// TIA Portal project "PLC and HMI project in TIA Portal.- simple" (V20)

(* hardware
DEVICE "S7-1200 station_1"  S7-1200 Station
   slot 0: "Rack_0"  S7-1200 Rack  Rack  V1.0
   slot 1: "PLC_1"  CPU 1212FC DC/DC/DC  6ES7 212-1AF40-0XB0  V4.7
DEVICE "HMI_1"  KTP700 Basic PN
   slot 0: "HMI_1"  KTP700 Basic PN  6AV2 123-2GB03-0AX0  17.0.0.0
   slot 1: "HMI_RT_1"  KTP700 Basic PN  6AV2 123-2GB03-0AX0  17.0.0.0
   slot 5: "HMI_1.IE_CP_1"  PROFINET Interface  17.0.0.0
      slot 1: "PROFINET Interface_1"  PROFINET Interface
         slot 1: "Port_1"  Port
*)

// ===== PLC "PLC_1"  CPU 1212FC DC/DC/DC =====

VAR_GLOBAL   // PLC tag table "Tag table_1"
   "Start_PB" AT %I0.0 : Bool;
   "Stop_PB" AT %M0.1 : Bool;
   "E_Stop" AT %M0.2 : Bool;
   "Conveyor_Motor" AT %Q0.0 : Bool;
END_VAR

DATA_BLOCK "Main_Safety_RTG1_DB"   // DB1, F_DB
{ S7_Optimized_Access := 'TRUE' }
NAME : FUSI
VERSION : 0.1
// stored: InstanceOfName Main_Safety_RTG1
"Main_Safety_RTG1"
BEGIN
END_DATA_BLOCK

FUNCTION_BLOCK "Main_Safety_RTG1"   // FB1, F_FBD
{ S7_Optimized_Access := 'TRUE' }
BEGIN
END_FUNCTION_BLOCK

ORGANIZATION_BLOCK "Main"   // OB1, LAD, ProgramCycle
TITLE = "Main Program Sweep (Cycle)"
{ S7_Optimized_Access := 'TRUE' }
VERSION : 0.1
   VAR_INPUT
      Initial_Call : Bool;   // Initial call of this OB
      Remanence : Bool;   // =True, if remanent data are available
   END_VAR
   VAR_TEMP   // added for the SCL form of the ladder/FBD networks
      _w1 : Bool;
   END_VAR
BEGIN

REGION Network 1
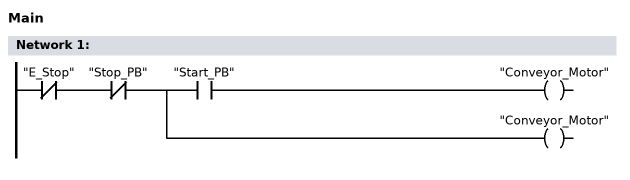
   RUNG wire#powerrail
      I_Contact( "E_Stop" )
      I_Contact( "Stop_PB" )
      wire#w1
      Contact( "Start_PB" )
      Coil( "Conveyor_Motor" )
   END_RUNG
   RUNG wire#w1
      Coil( "Conveyor_Motor" )
   END_RUNG
   // the same network as SCL:
   #_w1 := NOT "E_Stop" AND NOT "Stop_PB";
   "Conveyor_Motor" := #_w1 AND "Start_PB";
   "Conveyor_Motor" := #_w1;
END_REGION
END_ORGANIZATION_BLOCK

(* ===== HMI "HMI_RT_1" =====
system functions are stored by id; their names below are inferred from use
connection "HMI_Connection_1": ETHERNET, SMART_S7_1200_OMS

HMI tags "Default tag table"
   "Tag_ScreenNumber" : UInt, internal
   "Start_PB" : Bool = PLC Start_PB AT %I0.0, 1 s
   "Stop_PB" : Bool = PLC Stop_PB AT %M0.1, 1 s
   "E_Stop" : Bool = PLC E_Stop AT %M0.2, 1 s
   "Conveyor_Motor" : Bool = PLC Conveyor_Motor AT %Q0.0, 1 s

Template "Template_1" 800x480
   Button "Exit" at 714,429 size 71x50; TextOff 'Exit'; PictureOff "ExitRuntime_KTP700_Basic_PN_TR"; PictureOn "ExitRuntime_KTP700_Basic_PN_TR"
      on Release: StopRuntime(0)
   Button "Template_Button" at 614,429 size 71x50; TextOff 'Text'
   Button "Template_Button_1" at 514,429 size 71x50; TextOff 'Text'
   Button "Template_Button_2" at 414,429 size 71x50; TextOff 'Text'
   Button "Template_Button_3" at 314,429 size 71x50; TextOff 'Text'
   Button "Template_Button_4" at 214,429 size 71x50; TextOff 'Text'
   Button "Template_Button_5" at 114,429 size 71x50; TextOff 'Text'
   Button "Start screen" at 14,429 size 71x50; TextOff 'Start screen'; PictureOff "NavigateHome_KTP700_Basic_PN_TR"; PictureOn "NavigateHome_KTP700_Basic_PN_TR"
      on Release: ActivateScreen("Root screen", 0)
   SymbolicIOField "Symbolic_IO_Field_Screen" at 93,9 size 600x33; TextOff '0'; TextOn '1'; TextList "TextList_ScreenNames"
      ProcessValue <- "Tag_ScreenNumber"
      on Change: ActivateScreenByNumber("Tag_ScreenNumber", 0)
   DateTimeField "HmiScreenItemData" at 695,25 size 105x25
   DateTimeField "HmiScreenItemData_1" at 695,0 size 105x25
   GraphicView "Logo" at 0,0 size 91x51; Picture "Logo of HMI_1"

screen "Root screen" 800x480, template "Template_1"
   on GenerateScreen: SetTag("Stop_PB", 1)
   Button "Button_1" at 108,120 size 118x48; TextOff 'Start'
      on Click: SetBit("Start_PB")
      Appearance <- "Start_PB"
   Button "Button_2" at 293,119 size 123x48; TextOff 'Stop'
      on Click: SetBit("Stop_PB")
   Button "Button_3" at 481,120 size 123x48; TextOff 'Emmergency'
      on Click: SetBit("E_Stop")
   Circle "Circle_1" at 678,119 size 48x48
      Appearance <- "Conveyor_Motor"
   TextField "Text field_1" at 662,81 size 80x23; Text 'Motor On'
*)